// TIA Portal V20 export
DATA_BLOCK "BA010AZCRDR14_Stack1ConveyorAxisB"   // DB33, Motion_DB
// stored: InstanceOfName TO_SynchronousAxis, OfSystemLibElement TO_SynchronousAxis, OfSystemLibVersion 9.0
TO_SynchronousAxis   // technology object, version 9.0
// stored: Connection Interface Actor, InputAddress 51312, OutputAddress 51312
// stored: Connection Interface Sensor[1], InputAddress 51312, OutputAddress 51312, SensorIndexInActorTelegram 1
// stored: Connection Interface Torque, InputAddress 51472, OutputAddress 51472
// stored: SetPointCoupling Ref BA010AZCR_ConveyorVirtualAxis, Type TO_SynchronousAxis
   // // inherited from TO_PositioningAxis
   // // inherited from TO_SpeedAxis
   // // inherited from TO_Axis
   // // inherited from TO_Object
   // VAR
   //    Actor : TO_Struct_Actor;
   //    LoadGear : TO_Struct_LoadGear;
   //    DynamicLimits : TO_Struct_DynamicLimits;
   //    DynamicDefaults : TO_Struct_DynamicDefaults;
   // END_VAR
   // VAR
   //    Sensor : Array[1..4] of TO_Struct_Sensor;
   //    Mechanics : TO_Struct_Mechanics;
   //    PositionControl : TO_Struct_PositionControl;
   // END_VAR
   // VAR
   //    SynchronizedMotion { S7_SetPoint := 'True'} : TO_Struct_SynchronizedMotion;
   //    StatusSynchronizedMotion { ExternalWritable := 'False'; S7_SetPoint := 'True'} : TO_Struct_StatusSynchronizedMotion;
   // END_VAR
BEGIN
   Actor.DataAdaption := 1;
   Actor.Interface.AddressIn.RID := 16#208072a;
   Actor.Interface.AddressIn.AREA := 16#81;
   Actor.Interface.AddressIn.OFFSET := 51312;
   Actor.Interface.AddressOut.RID := 16#208072b;
   Actor.Interface.AddressOut.AREA := 16#82;
   Actor.Interface.AddressOut.OFFSET := 51312;
   Actor.Interface.EnableTorqueData := true;
   Actor.Interface.TorqueDataAddressIn.RID := 16#2080742;
   Actor.Interface.TorqueDataAddressIn.AREA := 16#81;
   Actor.Interface.TorqueDataAddressIn.OFFSET := 51472;
   Actor.Interface.TorqueDataAddressOut.RID := 16#2080743;
   Actor.Interface.TorqueDataAddressOut.AREA := 16#82;
   Actor.Interface.TorqueDataAddressOut.OFFSET := 51472;
   Actor.DriveParameter.ReferenceSpeed := 8000.0;
   Actor.DriveParameter.MaxSpeed := 1500.0;
   Actor.DriveParameter.ReferenceTorque := 8.74;
   LoadGear.Numerator := 10;
   DynamicLimits.MaxVelocity := 5000.0;
   DynamicLimits.MaxAcceleration := 100000.0;
   DynamicLimits.MaxDeceleration := 100000.0;
   DynamicLimits.MaxJerk := 2000000.0;
   DynamicDefaults.EmergencyDeceleration := 100000.0;
   Sensor[1]."Type" := 2;
   Sensor[1].DataAdaption := 1;
   Sensor[1].Interface.AddressIn.RID := 16#208072a;
   Sensor[1].Interface.AddressIn.AREA := 16#81;
   Sensor[1].Interface.AddressIn.OFFSET := 51312;
   Sensor[1].Interface.AddressOut.RID := 16#208072b;
   Sensor[1].Interface.AddressOut.AREA := 16#82;
   Sensor[1].Interface.AddressOut.OFFSET := 51312;
   Sensor[1].Parameter.DeterminableRevolutions := 4096;
   Mechanics.LeadScrew := 314.159265358979;
   PositionControl.EnableDSC := true;
   Actor.Interface.EnableTorqueData := True;
   _Actor.Interface.Telegram := 105;
   _Actor.DataAdaptionOffline := True;
   _Sensor[1].Interface.Telegram := 105;
   _Sensor[1].DataAdaptionOffline := True;
END_DATA_BLOCK
